{attribute 'hide_all_locals'}
FUNCTION_BLOCK AddMoverToGroupTask IMPLEMENTS ITask
VAR_INPUT
END_VAR
VAR_OUTPUT
END_VAR
VAR
	AddtoGrp			: MC_AddAxisToGroup;
	_caGroup			: REFERENCE TO AXES_GROUP_REF;
	_axis				: reference TO AXIS_REF;
	State: INT;
	_addMover : BOOL;
	_busy : BOOL;
	_error : BOOL;
	_done : BOOL;
	_moverNumber : UDINT;
END_VAR

CASE State OF
	0:
		IF _addMover THEN
			_done := FALSE;
			_error := FALSE;
			_busy := true;
			AddtoGrp.Execute := TRUE;
			IF AddtoGrp.Busy THEN
				State := 10;
				_addMover := FALSE;
			END_IF
		END_IF
	
	10:
		IF NOT AddtoGrp.Busy THEN
			IF AddtoGrp.Done THEN
				_done := TRUE;
			ELSIF AddtoGrp.Error THEN
				_error := TRUE;
			END_IF
			_busy := FALSE;
			AddtoGrp.Execute := false;
			State := 0;
		END_IF
END_CASE

AddtoGrp(AxesGroup := _caGroup,
			Axis := _axis,
			IdentInGroup := UDINT_TO_IDENTINGROUP(_moverNumber));

METHOD Abort : BOOL
AddtoGrp.Execute := FALSE;
Abort := true;
State := 0;
END_METHOD

METHOD AddMover : BOOL
VAR_INPUT
	MoverToAdd : IMover;
END_VAR
_axis REF= MoverToAdd.AxisRef;
_moverNumber := INT_TO_UDINT(MoverToAdd.IdentInGroup);
_busy := TRUE;
AddMover := _addMover := TRUE;
END_METHOD


PROPERTY Busy : BOOL
GET
Busy := _busy;
END_GET
END_PROPERTY


PROPERTY Done : BOOL
GET
Done := _done;
END_GET
END_PROPERTY


PROPERTY Error : BOOL
GET
Error := _error;
END_GET
END_PROPERTY

METHOD FB_init : BOOL
VAR_INPUT
	bInitRetains : BOOL; // if TRUE, the retain variables are initialized (warm start / cold start)
	bInCopyCode : BOOL;  // if TRUE, the instance afterwards gets moved into the copy code (online change)
	CAGroup : Reference TO AXES_GROUP_REF;	
END_VAR
_caGroup REF= CAGroup;
END_METHOD

END_FUNCTION_BLOCK

(* stored: Version 1.1.0.1, ProductVersion 3.1.4024.9
   POU AddMoverToGroupTask: Id {38d9c2dd-c50a-4b37-aa1d-638377a11576}, SpecialFunc None
   Method Abort: Id {d8ac89ea-7929-43cf-847c-ce36ce8ba2c8}
   Method AddMover: Id {b5d01066-95b3-4187-9840-17ba26e4ff68}
   Property Busy: Id {218184a8-dd89-4bad-8e2f-fc840856d81a}
   Get Get: Id {fc7f4575-ec7d-4ef2-8d11-dd9c112c4db2}
   Property Done: Id {25809c55-ac5a-4cf1-abb1-faea9e77608b}
   Get Get: Id {9011cbd7-cec9-4e7b-8d90-c54964a207f1}
   Property Error: Id {6f58c774-6cb9-4797-b38c-625ae7bdb7ed}
   Get Get: Id {bc46d96e-49ba-4622-8831-da4956773c11}
   Method FB_init: Id {c6af5b79-40e8-4ac6-b528-294ab1565185} *)
